# EPICS substitutions: iocs/bcur/iocBoot/iocbcur/substitutions/canberra_13.substitutions
file "$(MCA)/mcaApp/Db/simple_mca.db"
{
pattern
{P           M       DTYP           INP         PREC  CHANS}
{bcur:med:   mca1  "asynMCA"   "@asyn(AIM2/1 0)"    3  2048}
{bcur:med:   mca2  "asynMCA"   "@asyn(AIM2/1 1)"    3  2048}
{bcur:med:   mca3  "asynMCA"   "@asyn(AIM2/1 2)"    3  2048}
{bcur:med:   mca4  "asynMCA"   "@asyn(AIM2/2 0)"    3  2048}
{bcur:med:   mca5  "asynMCA"   "@asyn(AIM2/2 1)"    3  2048}
{bcur:med:   mca6  "asynMCA"   "@asyn(AIM2/2 2)"    3  2048}
{bcur:med:   mca7  "asynMCA"   "@asyn(AIM3/1 0)"    3  2048}
{bcur:med:   mca8  "asynMCA"   "@asyn(AIM3/1 1)"    3  2048}
{bcur:med:   mca9  "asynMCA"   "@asyn(AIM3/1 2)"    3  2048}
{bcur:med:   mca10 "asynMCA"   "@asyn(AIM3/2 0)"    3  2048}
{bcur:med:   mca11 "asynMCA"   "@asyn(AIM3/3 1)"    3  2048}
{bcur:med:   mca12 "asynMCA"   "@asyn(AIM3/4 2)"    3  2048}
{bcur:med:   mca13 "asynMCA"   "@asyn(AIM3/2 3)"    3  2048}
{bcur:med:   mca0  "Soft Channel"   ""     3  2048}
}

file "$(MCA)/mcaApp/Db/icb_amp.db"
{
pattern
{P			AMP		PORT}
{bcur:med:	amp1	"icbAmp1"}
{bcur:med:	amp2	"icbAmp2"}
{bcur:med:	amp3	"icbAmp3"}
{bcur:med:	amp4	"icbAmp4"}
{bcur:med:	amp5	"icbAmp5"}
{bcur:med:	amp6	"icbAmp6"}
{bcur:med:	amp7	"icbAmp7"}
{bcur:med:	amp8	"icbAmp8"}
{bcur:med:	amp9	"icbAmp9"}
{bcur:med:	amp10	"icbAmp10"}
{bcur:med:	amp11	"icbAmp11"}
{bcur:med:	amp12	"icbAmp12"}
{bcur:med:	amp13	"icbAmp13"}
}

file "$(MCA)/mcaApp/Db/icb_adc.db"
{
pattern
{P			ADC		PORT}
{bcur:med:	adc1	"icbAdc1"}
{bcur:med:	adc2	"icbAdc2"}
{bcur:med:	adc3	"icbAdc3"}
{bcur:med:	adc4	"icbAdc4"}
}

file "$(MCA)/mcaApp/Db/icb_hvps.db"
{
pattern
{P			HVPS	LIMIT	PORT}
{bcur:med:	hvps1	1000	"icbHvps1"}
}
